FUNCTION_BLOCK DigitalLamp_Wrapper
VAR
	IN AT%I* : BOOL;
	digitalLamp: OnOffDevice;
	_keyType: INT;		//	0: Tap/push button 1: Toggle/latch Button

	rtIN: R_TRIG;
	_app_TurnOn: BOOL;
	rt_app_TurnOn: R_TRIG;
	_app_TurnOff: BOOL;
	rt_app_TurnOff: R_TRIG;
	_app_TurnOnOff: BOOL;
	rt_app_TurnOnOff: R_TRIG;
END_VAR


	IF _keyType = 0 THEN
		rtIN(CLK:= IN, Q=> );
		rt_app_TurnOnOff(CLK:= _app_TurnOnOff, Q=> );
		
		IF rtIN.Q OR rt_app_TurnOnOff.Q THEN
			IF digitalLamp.Status = TRUE THEN
				digitalLamp.TurnOff();
			ELSE
				digitalLamp.TurnOn();	
			END_IF
		END_IF
		
		rt_app_TurnOn(CLK:= _app_TurnOn, Q=> );
		IF rt_app_TurnOn.Q THEN
			digitalLamp.TurnOn();
		END_IF
		rt_app_TurnOff(CLK:= _app_TurnOff, Q=> );
		IF rt_app_TurnOff.Q THEN
			digitalLamp.TurnOff();
		END_IF
		
	ELSIF _keyType = 1 THEN
		IF IN THEN
			digitalLamp.TurnOn();
		ELSE
			digitalLamp.TurnOff();
		END_IF
	ELSE
		digitalLamp.TurnOff();
	END_IF

PROPERTY App_TurnOff : BOOL
SET

	_app_TurnOff :=	App_TurnOff;
END_SET
END_PROPERTY

PROPERTY App_TurnOn : BOOL
SET

	_app_TurnOn :=	App_TurnOn;
END_SET
END_PROPERTY

PROPERTY App_TurnOnOff : BOOL
SET

	_app_TurnOnOff	:=	App_TurnOnOff;
END_SET
END_PROPERTY

PROPERTY KeyType : INT
SET

	_keyType	:=	KeyType;
END_SET
END_PROPERTY

END_FUNCTION_BLOCK

(* stored: Version 1.1.0.1, ProductVersion 3.1.4024.13
   POU DigitalLamp_Wrapper: Id {9b465ac5-45dd-4a22-82e9-cdd35cca90b9}, SpecialFunc None
   Property App_TurnOff: Id {86f9c277-8ea9-45a8-b666-ff0d965a146e}
   Set Set: Id {ef32cad1-c09b-4c54-85a2-dbfccbf7451c}
   Property App_TurnOn: Id {9a6b7db1-5d7f-4298-bc93-ad225917b945}
   Set Set: Id {270ee00b-43f4-4529-a384-5e848f0cc532}
   Property App_TurnOnOff: Id {3d78efad-7f45-4c12-8b1e-d24b3ea327f2}
   Set Set: Id {d916475e-8ca2-4f45-b157-a6aa24f17578}
   Property KeyType: Id {c5c90473-d7f9-4101-9598-80d9d7aaa278}
   Set Set: Id {95b50d8f-c9c0-41bd-8726-7977c5dab50c} *)
